FUNCTION_BLOCK FB_Area100 EXTENDS FB_ProgramBase
VAR_INPUT
END_VAR
VAR_OUTPUT
END_VAR
VAR
END_VAR

SUPER^();
// Management
	// Alarm management
	GVL_Area100.g_fbAlarmManager(i_bCmdResetFromHmi:= );
	
	// PackML status manager
	GVL_Area100.g_fbPackMLstatusManager();
	
	// Machine controls manager
	GVL_Area100.g_fbMachCtrlsManager(
		i_eCfgCtrlType				:= E_MachineControlsManager_Type.StartBtnAndStopBtnAndModeSelector,
		i_bReqStartBtnFromHmi		:= GVL_Area100.g_fbHmiMachCtrlsManager.q_bReqStart,
		i_bReqStopBtnFromHmi		:= GVL_Area100.g_fbHmiMachCtrlsManager.q_bReqStop,
		i_eReqModeFromHmi			:= GVL_Area100.g_fbHmiMachCtrlsManager.q_eReqMode,
		//i_astPackML_Status		:= , // Array entry set at unit
		i_nCfgNrOfUsedUnits			:= 1,
		i_stStackLightPackML_Status	:= GVL_Area100.g_unMachine100.q_stPackML_Status,
		i_bStaDownStream_NotRunning	:= ,
		i_bStaUpStream_NotRunning	:= ,
		i_bStaLowOnMaterials		:= );
	// Machine controls manager - HMI
	GVL_Area100.g_fbHmiMachCtrlsManager(
		i_itfModule	:= , 
		q_bReqStart	=> , 
		q_bReqStop	=> , 
		q_eReqMode	=> );

	
	
// Units
	// PLC units
	GVL_Area100.g_unMachine100(
		i_bReqEnable		:= TRUE, 
		i_bReqReset			:= GVL_Area100.g_fbAlarmManager.q_bCmdReset, 
		i_bReqSimulationOn	:= GVL.g_bCmdSimulationOn,
		i_stPackML_Command	:= GVL_Area100.g_fbMachCtrlsManager.q_stPackML_Command, 
		i_itfPackML_StatusManager	:= GVL_Area100.g_fbPackMLstatusManager,
		q_stPackML_Status	=> GVL_Area100.g_fbMachCtrlsManager.i_astPackML_Status[1]);
	
	// HMI units
	GVL_Area100.g_hmiUnMachine100(i_itfModule := GVL_Area100.g_unMachine100);

END_FUNCTION_BLOCK

(* stored: Version 1.1.0.1, ProductVersion 3.1.4024.10
   POU FB_Area100: Id {68d93498-5c7b-0e17-2bf9-5079bfd3f919}, SpecialFunc None *)
